// SIMATIC S7-200 project (STEP 7-Micro/WIN), CPU 224XP REL 02.01

ORGANIZATION_BLOCK MAIN:OB1
TITLE=PROGRAM COMMENTS
BEGIN
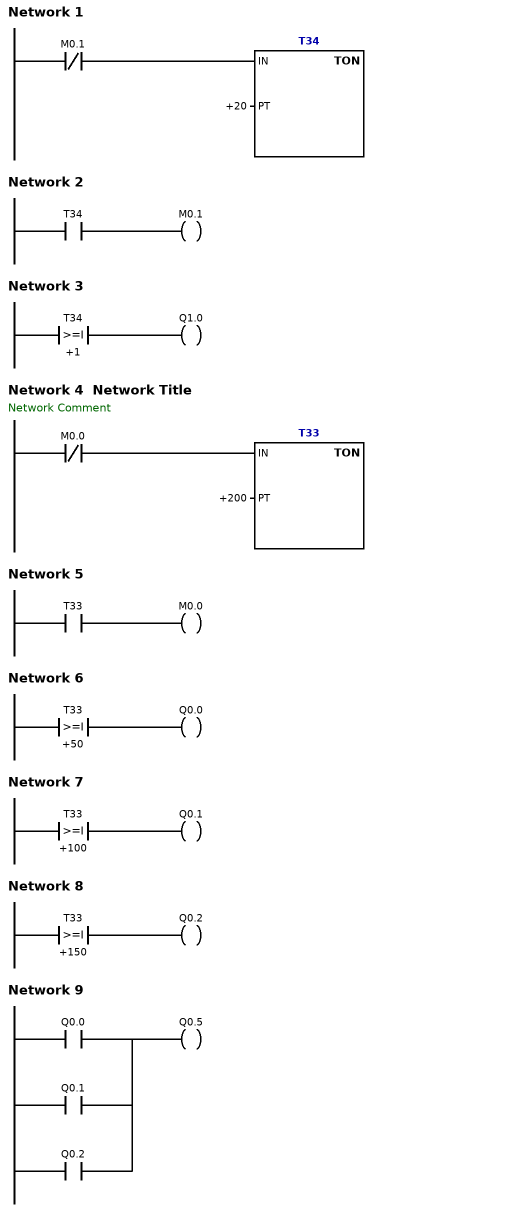
Network 1
LDN    M0.1
TON    T34, +20
Network 2
LD     T34
=      M0.1
Network 3
LDW>=  T34, +1
=      Q1.0
Network 4 // Network Title
// Network Comment
LDN    M0.0
TON    T33, +200
Network 5
LD     T33
=      M0.0
Network 6
LDW>=  T33, +50
=      Q0.0
Network 7
LDW>=  T33, +100
=      Q0.1
Network 8
LDW>=  T33, +150
=      Q0.2
Network 9
LD     Q0.0
O      Q0.1
O      Q0.2
=      Q0.5
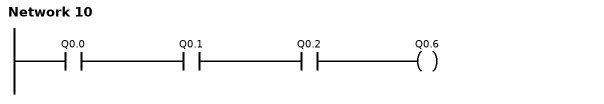
Network 10
LD     Q0.0
A      Q0.1
A      Q0.2
=      Q0.6
END_ORGANIZATION_BLOCK
